Staubli VAL3: Edit.pgx

program Edit(string x_sName)
  local bool l_bRes
  local num l_i
  local num l_nKey
  local num l_nRes
  local num l_nSelect
  local string l_sItem
  local string l_sValue
begin
  //edit the pallet
  cls()
  resize(sParameter,1,7)
  sParameter[0]="原点"
  sParameter[1]="X点"
  sParameter[2]="Y点"
  sParameter[3]="dX"
  sParameter[4]="dY"
  sParameter[5]="起点"
  sParameter[6]="工具"
  //
  resize(sListItemValue,1,size(sParameter))
  sListItemValue[0]=""
  sListItemValue[1]=""
  sListItemValue[2]=""
  sListItemValue[3]=toString(".3",uPallet[x_sName].ndX)
  sListItemValue[4]=toString(".3",uPallet[x_sName].ndY)
  sListItemValue[5]=""
  sListItemValue[6]=uPallet[sItem].sToolName

  //
  for l_i=0 to size(sParameter)-1
    call user:strlength(sParameter[l_i],user:nBottomX/2)
    l_sValue=sListItemValue[l_i]
    call user:strlength(l_sValue,user:nBottomX/2+1)
    sParameter[l_i]=sParameter[l_i]+":"+l_sValue
  endFor

  bUserRefresh=true
  bListRefresh=true
  nPage=1
  pPonit[0].trsf=uPallet[sItem].pO.trsf
  pPonit[1].trsf=uPallet[sItem].pX.trsf
  pPonit[2].trsf=uPallet[sItem].pY.trsf
  //
  do
    call Refresh()
    call user:setList(x_sName,sParameter,bUserRefresh,bListRefresh,nSelected,l_sItem,l_nKey)
    bUserRefresh=false
    bListRefresh=false
    call EnterPageKey(l_nKey,nSelected,sParameter[nSelected])
    delay(0)
  until l_nKey==255 or l_nKey==278
  //保存坐标系
  pPonit[0].trsf=uPallet[sItem].pO.trsf
  pPonit[1].trsf=uPallet[sItem].pX.trsf
  pPonit[2].trsf=uPallet[sItem].pY.trsf
  setFrame(pPonit[0],pPonit[1],pPonit[2],fFrame)
  //
  libSave()
  nPage=0
  bUserRefresh=true
  bListRefresh=true
end
